{attribute 'GeneratedUsingTerminal: EL6090-0000-0016'}
{attribute addProperty BoxType "EL6090-0000-0016"}
{attribute addProperty Id "StatusAT %I*Status_E3E7FD126"}
{attribute addProperty CRC "3773007075"}
{attribute addProperty Size "6"}
TYPE DIS_Inputs_E0E384E3 :
STRUCT
	{attribute addProperty Name "Status"}
	Status AT %I* : Status_E3E7FD12;
END_STRUCT
END_TYPE

(* stored: Version 1.2.0.0, ProductVersion 3.1.4024.9
   DUT DIS_Inputs_E0E384E3: Id {3818a9e0-40d5-4134-a0f0-0d7ef4cd9d13} *)
